FUNCTION F_2Norm : REAL
VAR_INPUT
	fA : REAL;
	fB : REAL;
END_VAR
VAR
END_VAR

F_2Norm := SQRT(fA*fA + fB*fB);

END_FUNCTION

(* stored: Version 1.1.0.1, ProductVersion 3.1.4024.12
   POU F_2Norm: Id {fa173772-ba73-4cf1-8b38-ecc044cf1fd4}, SpecialFunc None *)
